TYPE ST_BWK_Steuerung :
STRUCT
	Freigabe				: ST_Steuerung_auto_manu_BOOL;
	Freigabe_Deakt		: ST_Steuerung_auto_manu_BOOL;
	Betrieb_Anford		: ST_Steuerung_auto_manu_opti_BOOL;

	Regelung_Modus		: ST_Steuerung_auto_manu_opti_SINT;
	Regelung_Sollw		: ST_Steuerung_auto_manu_opti_REAL;

	Quittierung			: BOOL;
END_STRUCT
END_TYPE

(* stored: Version 1.1.0.1, ProductVersion 3.1.4024.9
   DUT ST_BWK_Steuerung: Id {684e0034-e212-4f0c-881d-3367ae310ced} *)
